{attribute 'GeneratedUsingTerminal: AT2040-0250-0022'}
{attribute addProperty BoxType "AT2040-0250-0022"}
{attribute addProperty Id "A_0107_AT2000_5233_0018_AT2000_5233AT2000_01D6DEDF80"}
{attribute addProperty CRC "2443323944"}
{attribute addProperty Size "80"}
TYPE A_0037_AT2040_0250_0022_91A22A28 EXTENDS AT2040_86175B41 :
STRUCT
	{attribute addProperty Name "A_0107_AT2000_5233_0018_AT2000_5233"}
	{attribute addProperty PreviousPort "A_0037(AT2040-0250-0022) : B"}
	A_0107_AT2000_5233_0018_AT2000_5233 : AT2000_01D6DEDF;
END_STRUCT
END_TYPE

(* stored: Version 1.2.0.0, ProductVersion 3.1.4024.9
   DUT A_0037_AT2040_0250_0022_91A22A28: Id {51f1be73-4d03-4164-92be-ea6315009e40} *)
